ADAPTER ADP_SERVICE_INFO (* Adapter Interface *)
  (* Standard: 61499-1 *)
  (* Version 0.0, 12/17/2022, Dmitrii, Flexbridge AB *)
  PACKAGE UAO.Hackathon;
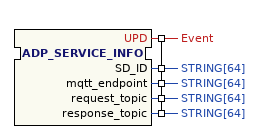
  EVENT_OUTPUT
    UPD WITH SD_ID, mqtt_endpoint, request_topic, response_topic; (* Request from Socket *)
  END_EVENT
  VAR_OUTPUT
    SD_ID : STRING[64]; (* Request Data from Socket *)
    mqtt_endpoint : STRING[64]; (* Response Data from Socket *)
    request_topic : STRING[64];
    response_topic : STRING[64];
  END_VAR
  SERVICE SOCKET/PLUG
    SEQUENCE request_confirm
      SOCKET.UPD(SD_ID) -> PLUG.UPD(SD_ID);
      PLUG.CNF(CNFD) -> SOCKET.CNF(CNFD);
    END_SEQUENCE
    SEQUENCE indication_response
      PLUG.IND(INDD) -> SOCKET.IND(INDD);
      SOCKET.RSP(mqtt_endpoint) -> PLUG.RSP(mqtt_endpoint);
    END_SEQUENCE
  END_SERVICE
END_ADAPTER
